KUKA KRL program: logoprog.src, logoprog.dat

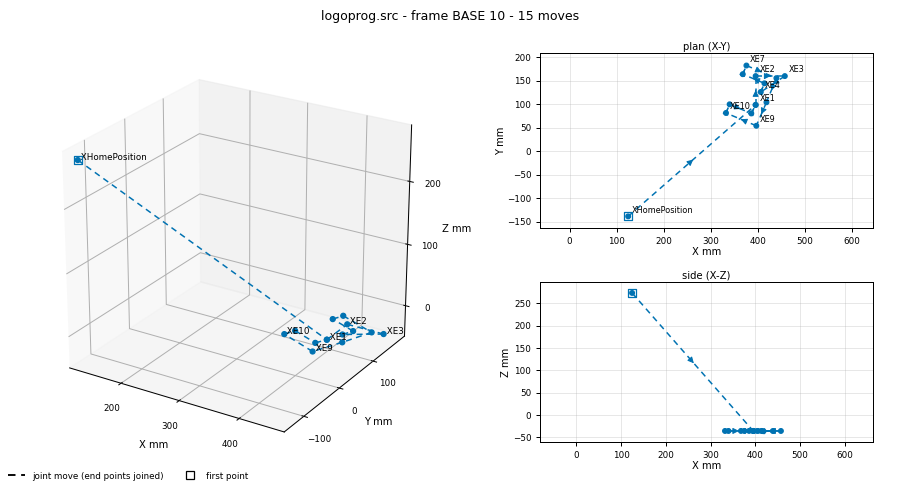
[picture p0: tool path of logoprog.src in frame BASE 10, 15 of 15 moves have a stored position in this frame; points joined in program order, loops and branches not executed]
--- logoprog.src ---
&ACCESS RVP
&REL 28
&PARAM EDITMASK = *
&PARAM TEMPLATE = C:\KRC\Roboter\Template\vorgabe
&PARAM DISKPATH = KRC:\R1\Program\Control Engineers\KZ_Prog
DEF LogoProg( )
  ;FOLD INI;%{PE}
    ;FOLD BASISTECH INI
      GLOBAL INTERRUPT DECL 3 WHEN $STOPMESS==TRUE DO IR_STOPM ( )
      INTERRUPT ON 3
      BAS (#INITMOV,0 )
    ;ENDFOLD (BASISTECH INI)
    ;FOLD USER INI
      ;Make your modifications here

    ;ENDFOLD (USER INI)
  ;ENDFOLD (INI)


  ;FOLD PTP HomePosition CONT Vel=100 % PDAT1 Tool[12]:CE_Marker Base[10]:baseCE;%{PE}%R 8.3.44,%MKUKATPBASIS,%CMOVE,%VPTP,%P 1:PTP, 2:HomePosition, 3:C_DIS, 5:100, 7:PDAT1
  $BWDSTART=FALSE
  PDAT_ACT=PPDAT1
  FDAT_ACT=FHomePosition
  BAS(#PTP_PARAMS,100)
  PTP XHomePosition C_DIS
  ;ENDFOLD

  ;FOLD PTP E1 CONT Vel=100 % PDAT1 Tool[12]:CE_Marker Base[10]:baseCE;%{PE}%R 8.3.44,%MKUKATPBASIS,%CMOVE,%VPTP,%P 1:PTP, 2:E1, 3:C_DIS, 5:100, 7:PDAT1
  $BWDSTART=FALSE
  PDAT_ACT=PPDAT1
  FDAT_ACT=FE1
  BAS(#PTP_PARAMS,100)
  PTP XE1 C_DIS
  ;ENDFOLD

  ;FOLD PTP E2 CONT Vel=100 % PDAT1 Tool[12]:CE_Marker Base[10]:baseCE;%{PE}%R 8.3.44,%MKUKATPBASIS,%CMOVE,%VPTP,%P 1:PTP, 2:E2, 3:C_DIS, 5:100, 7:PDAT1
  $BWDSTART=FALSE
  PDAT_ACT=PPDAT1
  FDAT_ACT=FE2
  BAS(#PTP_PARAMS,100)
  PTP XE2 C_DIS
  ;ENDFOLD

  ;FOLD PTP E3 CONT Vel=100 % PDAT1 Tool[12]:CE_Marker Base[10]:baseCE;%{PE}%R 8.3.44,%MKUKATPBASIS,%CMOVE,%VPTP,%P 1:PTP, 2:E3, 3:C_DIS, 5:100, 7:PDAT1
  $BWDSTART=FALSE
  PDAT_ACT=PPDAT1
  FDAT_ACT=FE3
  BAS(#PTP_PARAMS,100)
  PTP XE3 C_DIS
  ;ENDFOLD

  ;FOLD PTP E4 CONT Vel=100 % PDAT1 Tool[12]:CE_Marker Base[10]:baseCE;%{PE}%R 8.3.44,%MKUKATPBASIS,%CMOVE,%VPTP,%P 1:PTP, 2:E4, 3:C_DIS, 5:100, 7:PDAT1
  $BWDSTART=FALSE
  PDAT_ACT=PPDAT1
  FDAT_ACT=FE4
  BAS(#PTP_PARAMS,100)
  PTP XE4 C_DIS
  ;ENDFOLD
  ;FOLD PTP E5 CONT Vel=100 % PDAT1 Tool[12]:CE_Marker Base[10]:baseCE;%{PE}%R 8.3.44,%MKUKATPBASIS,%CMOVE,%VPTP,%P 1:PTP, 2:E5, 3:C_DIS, 5:100, 7:PDAT1
  $BWDSTART=FALSE
  PDAT_ACT=PPDAT1
  FDAT_ACT=FE5
  BAS(#PTP_PARAMS,100)
  PTP XE5 C_DIS
  ;ENDFOLD
  ;FOLD PTP E6 CONT Vel=100 % PDAT1 Tool[12]:CE_Marker Base[10]:baseCE;%{PE}%R 8.3.44,%MKUKATPBASIS,%CMOVE,%VPTP,%P 1:PTP, 2:E6, 3:C_DIS, 5:100, 7:PDAT1
  $BWDSTART=FALSE
  PDAT_ACT=PPDAT1
  FDAT_ACT=FE6
  BAS(#PTP_PARAMS,100)
  PTP XE6 C_DIS
  ;ENDFOLD
  ;FOLD PTP E7 CONT Vel=100 % PDAT1 Tool[12]:CE_Marker Base[10]:baseCE;%{PE}%R 8.3.44,%MKUKATPBASIS,%CMOVE,%VPTP,%P 1:PTP, 2:E7, 3:C_DIS, 5:100, 7:PDAT1
  $BWDSTART=FALSE
  PDAT_ACT=PPDAT1
  FDAT_ACT=FE7
  BAS(#PTP_PARAMS,100)
  PTP XE7 C_DIS
  ;ENDFOLD

  ;FOLD PTP E8 CONT Vel=100 % PDAT1 Tool[12]:CE_Marker Base[10]:baseCE;%{PE}%R 8.3.44,%MKUKATPBASIS,%CMOVE,%VPTP,%P 1:PTP, 2:E8, 3:C_DIS, 5:100, 7:PDAT1
  $BWDSTART=FALSE
  PDAT_ACT=PPDAT1
  FDAT_ACT=FE8
  BAS(#PTP_PARAMS,100)
  PTP XE8 C_DIS
  ;ENDFOLD

  ;FOLD PTP E15 CONT Vel=100 % PDAT1 Tool[12]:CE_Marker Base[10]:baseCE;%{PE}%R 8.3.44,%MKUKATPBASIS,%CMOVE,%VPTP,%P 1:PTP, 2:E15, 3:C_DIS, 5:100, 7:PDAT1
  $BWDSTART=FALSE
  PDAT_ACT=PPDAT1
  FDAT_ACT=FE15
  BAS(#PTP_PARAMS,100)
  PTP XE15 C_DIS
  ;ENDFOLD

  ;FOLD PTP E9 CONT Vel=100 % PDAT1 Tool[12]:CE_Marker Base[10]:baseCE;%{PE}%R 8.3.44,%MKUKATPBASIS,%CMOVE,%VPTP,%P 1:PTP, 2:E9, 3:C_DIS, 5:100, 7:PDAT1
  $BWDSTART=FALSE
  PDAT_ACT=PPDAT1
  FDAT_ACT=FE9
  BAS(#PTP_PARAMS,100)
  PTP XE9 C_DIS
  ;ENDFOLD

  ;FOLD PTP E10 CONT Vel=100 % PDAT1 Tool[12]:CE_Marker Base[10]:baseCE;%{PE}%R 8.3.44,%MKUKATPBASIS,%CMOVE,%VPTP,%P 1:PTP, 2:E10, 3:C_DIS, 5:100, 7:PDAT1
  $BWDSTART=FALSE
  PDAT_ACT=PPDAT1
  FDAT_ACT=FE10
  BAS(#PTP_PARAMS,100)
  PTP XE10 C_DIS
  ;ENDFOLD

  ;FOLD PTP E11 CONT Vel=100 % PDAT1 Tool[12]:CE_Marker Base[10]:baseCE;%{PE}%R 8.3.44,%MKUKATPBASIS,%CMOVE,%VPTP,%P 1:PTP, 2:E11, 3:C_DIS, 5:100, 7:PDAT1
  $BWDSTART=FALSE
  PDAT_ACT=PPDAT1
  FDAT_ACT=FE11
  BAS(#PTP_PARAMS,100)
  PTP XE11 C_DIS
  ;ENDFOLD

  ;FOLD PTP E12 CONT Vel=100 % PDAT1 Tool[12]:CE_Marker Base[10]:baseCE;%{PE}%R 8.3.44,%MKUKATPBASIS,%CMOVE,%VPTP,%P 1:PTP, 2:E12, 3:C_DIS, 5:100, 7:PDAT1
  $BWDSTART=FALSE
  PDAT_ACT=PPDAT1
  FDAT_ACT=FE12
  BAS(#PTP_PARAMS,100)
  PTP XE12 C_DIS
  ;ENDFOLD

  ;FOLD PTP E14 CONT Vel=100 % PDAT1 Tool[12]:CE_Marker Base[10]:baseCE;%{PE}%R 8.3.44,%MKUKATPBASIS,%CMOVE,%VPTP,%P 1:PTP, 2:E14, 3:C_DIS, 5:100, 7:PDAT1
  $BWDSTART=FALSE
  PDAT_ACT=PPDAT1
  FDAT_ACT=FE14
  BAS(#PTP_PARAMS,100)
  PTP XE14 C_DIS
  ;ENDFOLD

END

--- logoprog.dat ---
&ACCESS RVP
&REL 28
&PARAM EDITMASK = *
&PARAM TEMPLATE = C:\KRC\Roboter\Template\vorgabe
&PARAM DISKPATH = KRC:\R1\Program\Control Engineers\KZ_Prog
DEFDAT  LogoProg
;FOLD EXTERNAL DECLARATIONS;%{PE}%MKUKATPBASIS,%CEXT,%VCOMMON,%P
;FOLD BASISTECH EXT;%{PE}%MKUKATPBASIS,%CEXT,%VEXT,%P
EXT  BAS (BAS_COMMAND  :IN,REAL  :IN )
DECL INT SUCCESS
;ENDFOLD (BASISTECH EXT)
;FOLD USER EXT;%{E}%MKUKATPUSER,%CEXT,%VEXT,%P
;Make your modifications here

;ENDFOLD (USER EXT)
;ENDFOLD (EXTERNAL DECLARATIONS)
DECL BASIS_SUGG_T LAST_BASIS={POINT1[] "E15                     ",POINT2[] "E15                     ",CP_PARAMS[] "CPDAT0                  ",PTP_PARAMS[] "PDAT20                  ",CONT[] "C_DIS                   ",CP_VEL[] "2                       ",PTP_VEL[] "100                     ",SYNC_PARAMS[] "SYNCDAT                 ",SPL_NAME[] "S0                      ",A_PARAMS[] "ADAT0                   "}

DECL E6POS XHOMEPOSITION={X 124.580376,Y -138.145447,Z 273.274323,A 151.461227,B -2.73342681,C 156.499802,S 6,T 26,E1 0.0,E2 0.0,E3 0.0,E4 0.0,E5 0.0,E6 0.0}
DECL FDAT FHomePosition={TOOL_NO 12,BASE_NO 10,IPO_FRAME #BASE,POINT2[] " ",TQ_STATE FALSE}
DECL PDAT PPDAT1={VEL 100.000,ACC 100.000,APO_DIST 0.000,APO_MODE #CDIS,GEAR_JERK 50.0000,EXAX_IGN 0}

DECL E6POS XE1={X 395.5,Y 98.70,Z -35.3522224,A 142.888916,B -1.08895195,C 166.570938,S 6,T 26,E1 0.0,E2 0.0,E3 0.0,E4 0.0,E5 0.0,E6 0.0}
DECL FDAT FE1={TOOL_NO 12,BASE_NO 10,IPO_FRAME #BASE,POINT2[] " ",TQ_STATE FALSE}

DECL E6POS XE2={X 395.5,Y 160,Z -35.4037819,A 142.888916,B -1.08895195,C 166.570938,S 6,T 26,E1 0.0,E2 0.0,E3 0.0,E4 0.0,E5 0.0,E6 0.0}
DECL FDAT FE2={TOOL_NO 12,BASE_NO 10,IPO_FRAME #BASE,POINT2[] " ",TQ_STATE FALSE}

DECL E6POS XE3={X 457.5,Y 160,Z -35.4801979,A 142.888916,B -1.08895195,C 166.570938,S 6,T 26,E1 0.0,E2 0.0,E3 0.0,E4 0.0,E5 0.0,E6 0.0}
DECL FDAT FE3={TOOL_NO 12,BASE_NO 10,IPO_FRAME #BASE,POINT2[] " ",TQ_STATE FALSE}

DECL E6POS XE4={X 406.418701,Y 126.184174,Z -35.4049683,A 142.888916,B -1.08895195,C 166.570938,S 6,T 26,E1 0.0,E2 0.0,E3 0.0,E4 0.0,E5 0.0,E6 0.0}
DECL FDAT FE4={TOOL_NO 12,BASE_NO 10,IPO_FRAME #BASE,POINT2[] " ",TQ_STATE FALSE}

DECL E6POS XE5={X 414.183502,Y 144.615082,Z -35.4078712,A 142.888916,B -1.08895195,C 166.570938,S 6,T 26,E1 0.0,E2 0.0,E3 0.0,E4 0.0,E5 0.0,E6 0.0}
DECL FDAT FE5={TOOL_NO 12,BASE_NO 10,IPO_FRAME #BASE,POINT2[] " ",TQ_STATE FALSE}

DECL E6POS XE6={X 368.119141,Y 164.020,Z -35.3868637,A 142.888916,B -1.08895195,C 166.570938,S 6,T 26,E1 0.0,E2 0.0,E3 0.0,E4 0.0,E5 0.0,E6 0.0}
DECL FDAT FE6={TOOL_NO 12,BASE_NO 10,IPO_FRAME #BASE,POINT2[] " ",TQ_STATE FALSE}

DECL E6POS XE7={X 375.883972,Y 182.450912,Z -35.3897667,A 142.888916,B -1.08895195,C 166.570938,S 6,T 26,E1 0.0,E2 0.0,E3 0.0,E4 0.0,E5 0.0,E6 0.0}
DECL FDAT FE7={TOOL_NO 12,BASE_NO 10,IPO_FRAME #BASE,POINT2[] " ",TQ_STATE FALSE}

DECL E6POS XE8={X 439.590698,Y 155.614014,Z -35.5337158,A 142.888916,B -1.08895195,C 166.570938,S 6,T 26,E1 0.0,E2 0.0,E3 0.0,E4 0.0,E5 0.0,E6 0.0}
DECL FDAT FE8={TOOL_NO 12,BASE_NO 10,IPO_FRAME #BASE,POINT2[] " ",TQ_STATE FALSE}


DECL E6POS XE9={X 396.940277,Y 54.4040375,Z -35.5569534,A 142.888916,B -1.08895183,C 166.570938,S 6,T 26,E1 0.0,E2 0.0,E3 0.0,E4 0.0,E5 0.0,E6 0.0}
DECL FDAT FE9={TOOL_NO 12,BASE_NO 10,IPO_FRAME #BASE,POINT2[] " ",TQ_STATE FALSE}

DECL E6POS XE10={X 332.431854,Y 81.5786667,Z -35.4574165,A 142.888916,B -1.08895183,C 166.570938,S 6,T 26,E1 0.0,E2 0.0,E3 0.0,E4 0.0,E5 0.0,E6 0.0}
DECL FDAT FE10={TOOL_NO 12,BASE_NO 10,IPO_FRAME #BASE,POINT2[] " ",TQ_STATE FALSE}

DECL E6POS XE11={X 340.196686,Y 100.009567,Z -35.4503212,A 142.888916,B -1.08895183,C 166.570938,S 6,T 26,E1 0.0,E2 0.0,E3 0.0,E4 0.0,E5 0.0,E6 0.0}
DECL FDAT FE11={TOOL_NO 12,BASE_NO 10,IPO_FRAME #BASE,POINT2[] " ",TQ_STATE FALSE}

DECL E6POS XE12={X 386.274139,Y 80.5991211,Z -35.3514175,A 142.888916,B -1.08895183,C 166.570938,S 6,T 26,E1 0.0,E2 0.0,E3 0.0,E4 0.0,E5 0.0,E6 0.0}
DECL FDAT FE12={TOOL_NO 12,BASE_NO 10,IPO_FRAME #BASE,POINT2[] " ",TQ_STATE FALSE}

DECL E6POS XE13={X 395.462067,Y 98.7066498,Z -35.3522224,A 142.888916,B -1.08895195,C 166.570938,S 6,T 26,E1 0.0,E2 0.0,E3 0.0,E4 0.0,E5 0.0,E6 0.0}
DECL FDAT FE13={TOOL_NO 12,BASE_NO 10,IPO_FRAME #BASE,POINT2[] " ",TQ_STATE FALSE}

DECL E6POS XE14={X 395.462067,Y 98.7066498,Z -35.3522224,A 142.888916,B -1.08895195,C 166.570938,S 6,T 26,E1 0.0,E2 0.0,E3 0.0,E4 0.0,E5 0.0,E6 0.0}
DECL FDAT FE14={TOOL_NO 12,BASE_NO 10,IPO_FRAME #BASE,POINT2[] " ",TQ_STATE FALSE}

DECL E6POS XE15={X 418.492371,Y 104.338318,Z -35.9924,A 142.889404,B -1.08916330,C 166.571503,S 6,T 26,E1 0.0,E2 0.0,E3 0.0,E4 0.0,E5 0.0,E6 0.0}
DECL FDAT FE15={TOOL_NO 12,BASE_NO 10,IPO_FRAME #BASE,POINT2[] " ",TQ_STATE FALSE}
ENDDAT
